FUNCTION_BLOCK EL3681
VAR
	_io : EL3681_Data;
	{attribute addProperty Name "WcState"}
	_wcState : WcStateInputToggle;
	{attribute addProperty Name "Info data"}
	_infoData : InfoDataAds;
END_VAR

PROPERTY IO : REFERENCE TO EL3681_Data
GET
IO REF= _io;
END_GET
END_PROPERTY

PROPERTY WcState : REFERENCE TO WcStateInputToggle
GET
WcState REF= _wcState;
END_GET
END_PROPERTY

END_FUNCTION_BLOCK

(* stored: Version 1.1.0.1, ProductVersion 3.1.4024.9
   POU EL3681: Id {116a7d95-e460-0cd0-3875-4d33af3113a4}, SpecialFunc None
   Property IO: Id {d2da3589-fc82-08fb-324d-431839bc5429}
   Get Get: Id {e05e0be7-5736-0cb0-3ae5-f36d2995ac4f}
   Property WcState: Id {085c2436-1173-07cc-3886-5f1dceafd5e2}
   Get Get: Id {8bc5419b-f2db-0368-2264-58de25464f73} *)
